FUNCTION_BLOCK FB_Dispenser
VAR_INPUT
	bEnable : BOOL;
	bExecute : BOOL;
	rDistance : REAL;
	
END_VAR
VAR_OUTPUT
	eState : eBetriebszustand;
END_VAR
VAR
	mcReset : MC_Reset;
	mcPower : MC_Power;
	mcMoveRelative : MC_MoveRelative;
	nState : INT;
END_VAR

VAR_IN_OUT
	// Achsen Ref
	ax : Axis_Ref;
END_VAR

ax.ReadStatus();

mcReset(
	Axis:= ax, 
	Execute:= , 
	Done=> , 
	Busy=> , 
	Error=> , 
	ErrorID=> );

mcPower(
	Axis:= ax, 
	Enable:= , 
	Enable_Positive:= , 
	Enable_Negative:= , 
	Override:= , 
	BufferMode:= , 
	Options:= , 
	Status=> , 
	Busy=> , 
	Error=> , 
	ErrorID=> );
	
mcMoveRelative(
	Axis:= ax, 
	Execute:= , 
	Distance:= 10, 
	Velocity:= , 
	Acceleration:= , 
	Deceleration:= , 
	Jerk:= , 
	BufferMode:= , 
	Options:= , 
	Done=> , 
	Busy=> , 
	Active=> , 
	CommandAborted=> , 
	Error=> , 
	ErrorID=> );
	
IF NOT mcPower.Status THEN
	nState := 0;
END_IF

CASE nState OF
	0: // OFF
	eState := eBetriebszustand.Off;
	mcPower.Enable := TRUE;
	mcPower.Enable_Positive := TRUE;
	IF bEnable AND mcPower.Status THEN
		nState := 20; //Ready
	ELSIF bEnable AND NOT mcPower.Status THEN
		nState := 10; // Init-Rest
	END_IF
	
	
	10: // Init - Reset
	eState := eBetriebszustand.Init;
	mcReset.Execute := TRUE;
	mcPower.Enable := FALSE;
	IF mcReset.Done THEN
		mcReset.Execute := FALSE;
		nState := 11;
	END_IF
	
	11: // Init - Power
	eState := eBetriebszustand.Init;
	mcPower.Enable := TRUE;
	mcReset.Execute := FALSE;
	IF mcPower.Status THEN
		nState := 20;
	END_IF
	
	20: //Ready
	eState := eBetriebszustand.Ready;
	IF bExecute THEN
		nState := 30;
	END_IF
	
	30: //Production
	eState := eBetriebszustand.Production;
	mcMoveRelative.Execute := TRUE;
	mcMoveRelative.Velocity := 20;
	mcMoveRelative.Acceleration := 20;
	mcMoveRelative.Distance := rDistance;
	
	IF mcMoveRelative.Done THEN
		nState := 40;
	END_IF
	
	40: // Fertig
	eState := eBetriebszustand.Done;
	mcMoveRelative.Execute := FALSE;
	
	IF NOT bExecute THEN
		nState := 20;
	END_IF
END_CASE

END_FUNCTION_BLOCK

(* stored: Version 1.1.0.1, ProductVersion 3.1.4024.15
   POU FB_Dispenser: Id {b6e3b9f0-d31f-4bd1-a392-726175ee30d8}, SpecialFunc None *)
